// TIA Portal V19 export
TYPE "LEXCHANGETRAY_typeAxisSimpleControlNodeMonitoring_2"
// stored: Access Published
   STRUCT
      valid { ExternalWritable := 'False'} : Bool := FALSE;   // Valid set of output values available at the FB
      busy { ExternalWritable := 'False'} : Bool := FALSE;   // Working and new output values can be expected
      error { ExternalWritable := 'False'} : Bool := FALSE;   // An error occurred during the execution of the FB
      status { ExternalWritable := 'False'} : Word := 16#7000;   // 16#0000-16#7FFF: Status of the FB; 16#8000-16#FFFF: Error identification
      subfunctionStatus { ExternalWritable := 'False'} : Word := 16#0000;   // Status or return value of called FBs, FCs, system blocks or other status information
      axisEnabled { ExternalWritable := 'False'} : Bool := FALSE;   // TRUE: Axis is enabled. Motion commands can be executed
      resetDone { ExternalWritable := 'False'} : Bool := FALSE;   // TRUE: Technology alarms have been acknowledged or reinitialization has been executed
      resetBusy { ExternalWritable := 'False'} : Bool := FALSE;   // TRUE: Reset or reinitialization is being processed
      resetAborted { ExternalWritable := 'False'} : Bool := FALSE;   // TRUE: Reset or reinitialization was aborted by another command
      homeDone { ExternalWritable := 'False'} : Bool := FALSE;   // TRUE: Homing completed without error
      homeBusy { ExternalWritable := 'False'} : Bool := FALSE;   // TRUE: Homing is being processed
      homeAborted { ExternalWritable := 'False'} : Bool := FALSE;   // TRUE: Homing was aborted by another command
      haltDone { ExternalWritable := 'False'} : Bool := FALSE;   // MC_Halt: Job is completed / TRUE: Velocity zero has been reached
      haltBusy { ExternalWritable := 'False'} : Bool := FALSE;   // MC_Halt: Job is running / TRUE: Axis is braking
      haltAborted { ExternalWritable := 'False'} : Bool := FALSE;   // TRUE: Braking was aborted by another command
      posAbsoluteDone { ExternalWritable := 'False'} : Bool := FALSE;   // TRUE: The target position has been reached
      posAbsoluteBusy { ExternalWritable := 'False'} : Bool := FALSE;   // TRUE: Absolute positioning is being processed
      posAbsoluteAborted { ExternalWritable := 'False'} : Bool := FALSE;   // TRUE: Absolute positioning was aborted by another command
      posRelativeDone { ExternalWritable := 'False'} : Bool := FALSE;   // TRUE: The target position has been reached
      posRelativeBusy { ExternalWritable := 'False'} : Bool := FALSE;   // TRUE: Relative positioning is being processed
      posRelativeAborted { ExternalWritable := 'False'} : Bool := FALSE;   // TRUE: Relative positioning was aborted by another command
      inVelocity { ExternalWritable := 'False'} : Bool := FALSE;   // TRUE: The velocity setpoint/speed setpoint has been reached
      moveVelocityBusy { ExternalWritable := 'False'} : Bool := FALSE;   // TRUE: Axis is accelerating/decelerating to reach velocity setpoint/speed setpoint
      moveVolocityAborted { ExternalWritable := 'False'} : Bool := FALSE;   // TRUE: Constant velocity/speed was aborted by another command
      jogInVelocity { ExternalWritable := 'False'} : Bool := FALSE;   // MC_MoveJog: The velocity setpoint / speed setpoint was reached and will be maintained / TRUE: The velocity setpoint/speed setpoint has been reached
      jogBusy { ExternalWritable := 'False'} : Bool := FALSE;   // MC_MoveJog: Job is running / TRUE: Axis is jogging
      jogAborted { ExternalWritable := 'False'} : Bool := FALSE;   // TRUE: Jogging was aborted by another command
      torqueBusy : Bool;
      InClamping : Bool;
      InLimitation : Bool;
      stopDone { ExternalWritable := 'False'} : Bool := FALSE;   // TRUE: Axis has reached standstill
      stopBusy { ExternalWritable := 'False'} : Bool := FALSE;   // TRUE: Axis is braking to a standstill
      stopAborted { ExternalWritable := 'False'} : Bool := FALSE;   // TRUE: Stopping was aborted by another command
      axisType { ExternalWritable := 'False'} : UDInt := 0;   // 0: unknown; 1:TO_PositioningAxis; 2: TO_SpeedAxis; 3: TO_SynchronousAxis; 4: Reserved; 5: TO_ExternalEncoder
      statusWord { ExternalWritable := 'False'} : "LBC_typeAxisSimpleControlStatusWord";   // Status information of the TO
      warningWord { ExternalWritable := 'False'} : "LBC_typeAxisSimpleControlWarningWord";   // Warnings of the TO
      errorWord { ExternalWritable := 'False'} : "LBC_typeAxisSimpleControlErrorWord";   // Errors of the TO
      errorNumber { ExternalWritable := 'False'} : UDInt := 0;   // Technology alarm number
      errorReaction { ExternalWritable := 'False'} : DInt := 0;   // Effective alarm response (0: no reaction; 1: stop with current dynamic values; 2: stop with maximum dynamic values; 3: stop with emergency stop ramp; 4: remove enable; 5: track setpoints); external encoder (0: no reaction; 10: remove enable)
      position { ExternalWritable := 'False'} : LReal := 0.0;   // Position setpoint
      velocity { ExternalWritable := 'False'} : LReal := 0.0;   // Velocity setpoint / speed setpoint
      actualPosition { ExternalWritable := 'False'} : LReal := 0.0;   // Actual position
      actualVelocity { ExternalWritable := 'False'} : LReal := 0.0;   // Actual velocity
      actualTorque : LReal;
      targetPosition { ExternalWritable := 'False'} : LReal := 0.0;   // Target position
      followingError { ExternalWritable := 'False'} : LReal := 0.0;   // Current following error
      lengthUnit { ExternalWritable := 'False'} : UDInt := 0;   // Unit for position (1004=rad, 1005=°, 1010=m, 1011=km, 1013=mm, 1014=µm, 1015=nm, 1018=ft, 1019=in, 1021=mi); with high resolution (1536=mm, 1537=°)
      velocityUnit { ExternalWritable := 'False'} : UDInt := 0;   // Unit for velocity (1061=m/s, 1062=mm/s, 1063=m/h 1064=km/h, 1066=in/s, 1067=ft/s, 1069=in/min, 1070=ft/min, 1075=mi/h, 1082=1/s, 1083=1/min, 1086=rad/s, 1521=°/s, 1522=°/min, 1523=rad/min, 1524=mm/min, 1525=m/min, 1526=mm/h, 1527=km/min, 1528=1/h); with high resolution (1538=mm/s, 1539=°/s)
   END_STRUCT;
END_TYPE
